// Implicitly generated code : DO NOT EDIT
FUNCTION CheckBounds : DINT
VAR_INPUT
	index, lower, upper: DINT;
END_VAR

// Implicitly generated code : Only an Implementation suggestion
IF  index < lower THEN
	CheckBounds := lower;
	gvlChecks.dCheckBounds := gvlChecks.dCheckBounds + 1;
ELSIF  index > upper THEN
	CheckBounds := upper;
	gvlChecks.dCheckBounds := gvlChecks.dCheckBounds + 1;
ELSE  
	CheckBounds := index;
END_IF

END_FUNCTION

(* stored: Version 1.1.0.1, ProductVersion 3.1.4026.13, FileIdentifier a0b73508612ee5c0b9a1c663ba5db9e27b35be8a, FileSignature 822b599e29b9230cf05873bf64e1b4a8f621a8aa602429affebc2aba2bfaed9a3955aaf078fb2a3403ea0da7042da1801e327df2970372a2ea795a7ead8746b44a16efb5d52e45a618f937fa17c371ba06dc0ad8e335c89ac85b00e22fcd26353feb2efca2a2c93d8a5b3ed14fdc622f455452659054b67e7c1e3e234e7ba09980e2f6638642becc99e0bd974a6514e98998468bcb86c0c23c9a849285c8070ac5607b5474ece09d101c20b7df3f19ef732098140d00173b255115f44cb478a7accc8e145ab0c5d3d4240127e664b8d2fa8514089292ccfa02bb18e60624c5c39221c599de2fcd13f9df05d6c4b3da954fe5b19d46a2eb25dd2e43a65f9f915d
   POU CheckBounds: Id {a2917252-a5bd-462b-898a-66626a9a5ae1}, SpecialFunc CheckBounds *)
